# EPICS substitutions: current/app/Db/AnalogInputs.substitutions
file hpm900ai.template {
  pattern
  {RECORD_NAME, OFFSET, DESC}
  {HPT:1:AI_RBV, 5, "Card 1 Channel 0 Analog Input HPT-1"}
  {LPT:1:AI_RBV, 6, "Card 1 Channel 1 Analog Input LPT-1"}
  {VPT:1:AI_RBV, 7, "Card 1 Channel 2 Analog Input VPT-1"}
  {HPT:2:AI_RBV, 8, "Card 1 Channel 3 Analog Input HPT-2"}
  {LPT:2:AI_RBV, 9, "Card 1 Channel 3 Analog Input LPT-2"}
  {VPT:2:AI_RBV, 10, "Card 1 Channel 5 Analog Input VPT-2"}
  {LPT:3:AI_RBV, 11, "Card 1 Channel 6 Analog Input LPT-3"}
}
